// Mitsubishi GX Works2 project: 세척,열풍건조, 동결건조(최신화)   PLC: Q02U

PROGRAM INPUT
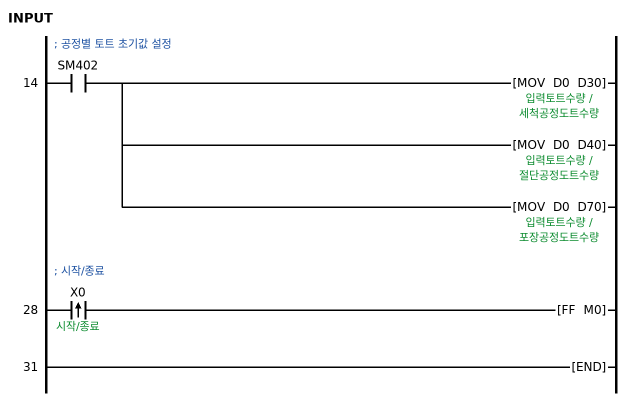
; 공정별 토트 초기값 설정
14    LD      SM402
      MOV     D0 D30  ; 입력토트수량 / 세척공정도트수량
      MOV     D0 D40  ; 절단공정도트수량
      MOV     D0 D70  ; 포장공정도트수량
; 시작/종료
28    LDP     X0  ; 시작/종료
      FF      M0
31    END
END_PROGRAM

PROGRAM 세척공정
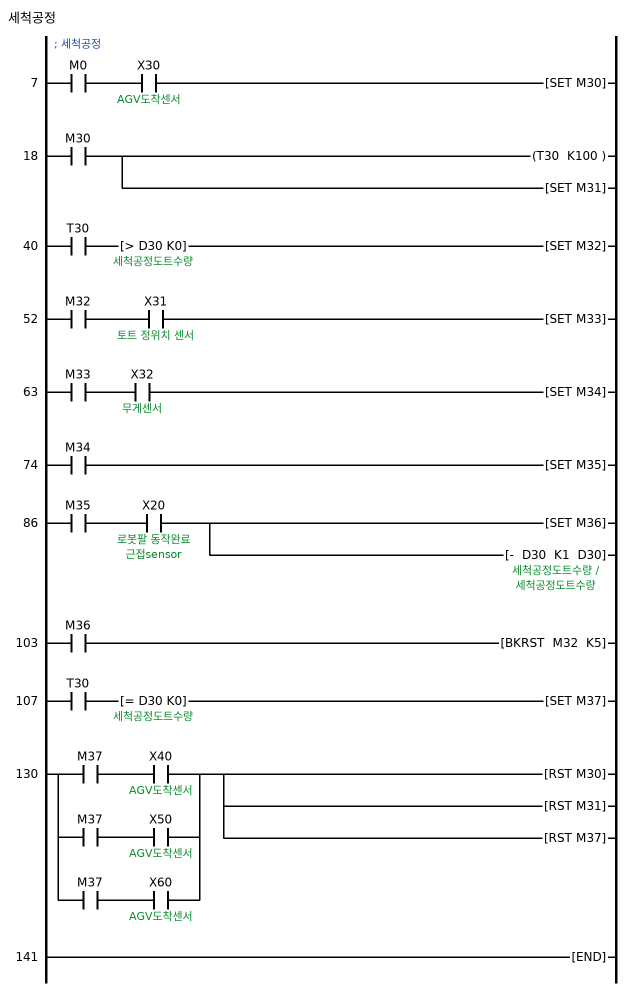
; 세척공정
7     LD      M0
      AND     X30  ; AGV도착센서
      SET     M30
        [note] 펌프모터 ON
18    LD      M30
      OUT     T30 K100
        [note] 펌핑모터 OFF
      SET     M31
        [note] SubCVY ON
40    LD      T30
      AND>    D30 K0  ; 세척공정도트수량
      SET     M32
        [note] 토트 발생
52    LD      M32
      AND     X31  ; 토트 정위치 센서
      SET     M33
        [note] MainCVY ON
63    LD      M33
      AND     X32  ; 무게센서
      SET     M34
        [note] MAinCVY OFF
74    LD      M34
      SET     M35
        [note] 하역 로봇팔 ON
86    LD      M35
      AND     X20  ; 로봇팔 동작완료 근접sensor
      SET     M36
        [note] 하역 로봇팔 OFF
      -       D30 K1 D30
103   LD      M36
      BKRST   M32 K5
107   LD      T30
      AND=    D30 K0  ; 세척공정도트수량
      SET     M37
        [note] AGV 다음 공정 이동, SubCVY OFF
130   LD      M37
      AND     X40  ; AGV도착센서
      LD      M37
      AND     X50  ; AGV도착센서
      ORB
      LD      M37
      AND     X60  ; AGV도착센서
      ORB
      RST     M30
      RST     M31
      RST     M37
141   END
END_PROGRAM

PROGRAM 열풍건조
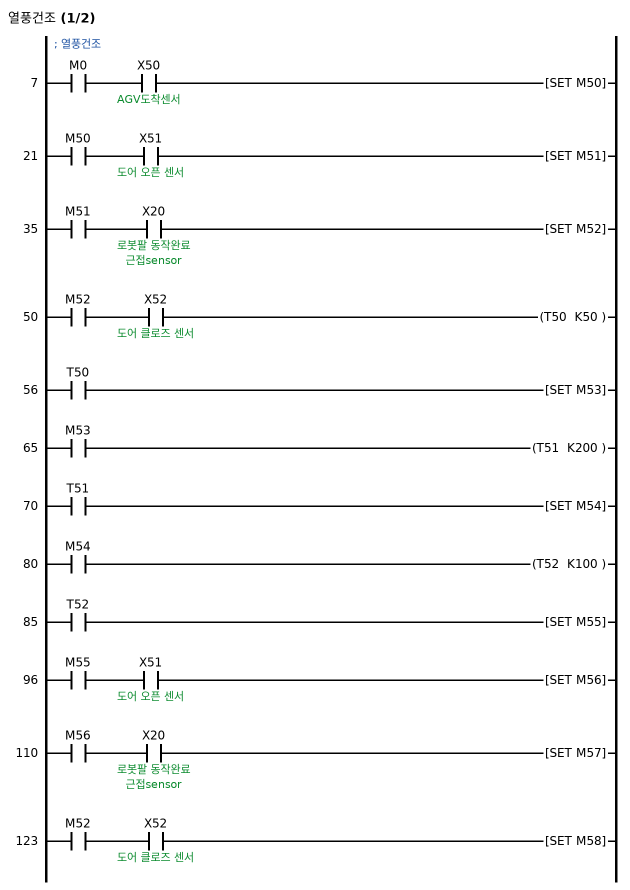
; 열풍건조
7     LD      M0
      AND     X50  ; AGV도착센서
      SET     M50
        [note] 도어 오픈모터(정)
21    LD      M50
      AND     X51  ; 도어 오픈 센서
      SET     M51
        [note] 상역 로봇 팔동작
35    LD      M51
      AND     X20  ; 로봇팔 동작완료 근접sensor
      SET     M52
        [note] 도어 클로즈모터(정)
50    LD      M52
      AND     X52  ; 도어 클로즈 센서
      OUT     T50 K50
56    LD      T50
      SET     M53
        [note] 건조기 ON
65    LD      M53
      OUT     T51 K200
70    LD      T51
      SET     M54
        [note] 건조기 OFF
80    LD      M54
      OUT     T52 K100
85    LD      T52
      SET     M55
        [note] 도어 오픈CYL
96    LD      M55
      AND     X51  ; 도어 오픈 센서
      SET     M56
        [note] 하역 로봇팔 동작
110   LD      M56
      AND     X20  ; 로봇팔 동작완료 근접sensor
      SET     M57
        [note] 도어 클로즈CYL
123   LD      M52
      AND     X52  ; 도어 클로즈 센서
      SET     M58
        [note] AGV 다음 공정 이동
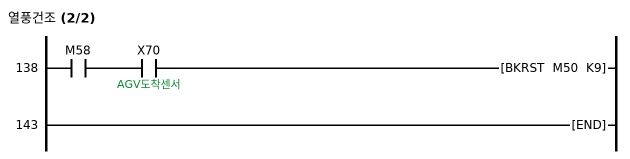
138   LD      M58
      AND     X70  ; AGV도착센서
      BKRST   M50 K9
143   END
END_PROGRAM

PROGRAM OUTPUT
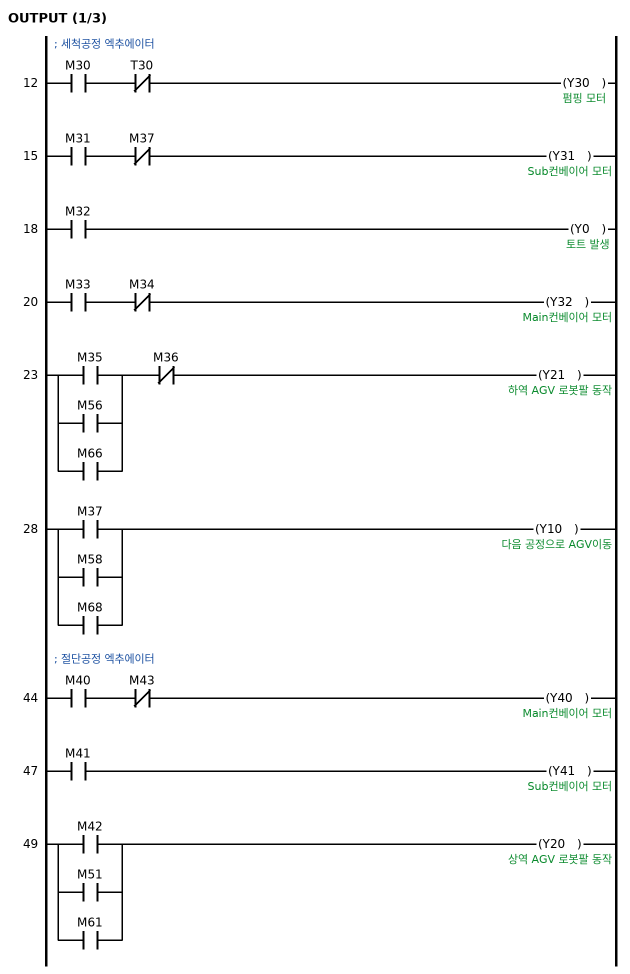
; 세척공정 엑추에이터
12    LD      M30
      ANI     T30
      OUT     Y30  ; 펌핑 모터
15    LD      M31
      ANI     M37
      OUT     Y31  ; Sub컨베이어 모터
18    LD      M32
      OUT     Y0  ; 토트 발생
20    LD      M33
      ANI     M34
      OUT     Y32  ; Main컨베이어 모터
23    LD      M35
      OR      M56
      OR      M66
      ANI     M36
      OUT     Y21  ; 하역 AGV 로봇팔 동작
28    LD      M37
      OR      M58
      OR      M68
      OUT     Y10  ; 다음 공정으로 AGV이동
; 절단공정 엑추에이터
44    LD      M40
      ANI     M43
      OUT     Y40  ; Main컨베이어 모터
47    LD      M41
      OUT     Y41  ; Sub컨베이어 모터
49    LD      M42
      OR      M51
      OR      M61
      OUT     Y20  ; 상역 AGV 로봇팔 동작
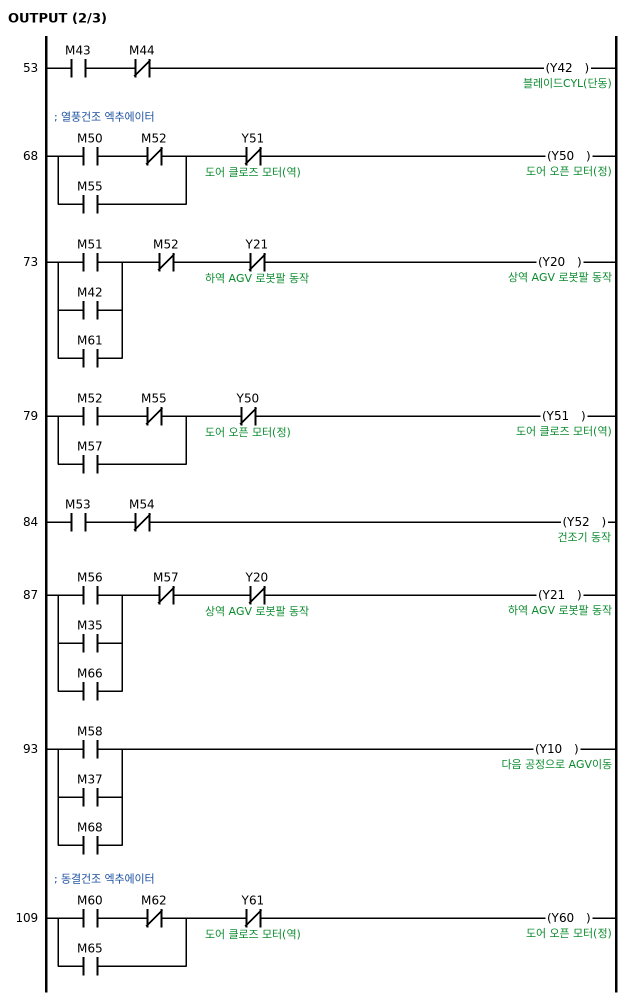
53    LD      M43
      ANI     M44
      OUT     Y42  ; 블레이드CYL(단동)
; 열풍건조 엑추에이터
68    LD      M50
      ANI     M52
      OR      M55
      ANI     Y51  ; 도어 클로즈 모터(역)
      OUT     Y50  ; 도어 오픈 모터(정)
73    LD      M51
      OR      M42
      OR      M61
      ANI     M52
      ANI     Y21  ; 하역 AGV 로봇팔 동작
      OUT     Y20  ; 상역 AGV 로봇팔 동작
79    LD      M52
      ANI     M55
      OR      M57
      ANI     Y50  ; 도어 오픈 모터(정)
      OUT     Y51  ; 도어 클로즈 모터(역)
84    LD      M53
      ANI     M54
      OUT     Y52  ; 건조기 동작
87    LD      M56
      OR      M35
      OR      M66
      ANI     M57
      ANI     Y20  ; 상역 AGV 로봇팔 동작
      OUT     Y21  ; 하역 AGV 로봇팔 동작
93    LD      M58
      OR      M37
      OR      M68
      OUT     Y10  ; 다음 공정으로 AGV이동
; 동결건조 엑추에이터
109   LD      M60
      ANI     M62
      OR      M65
      ANI     Y61  ; 도어 클로즈 모터(역)
      OUT     Y60  ; 도어 오픈 모터(정)
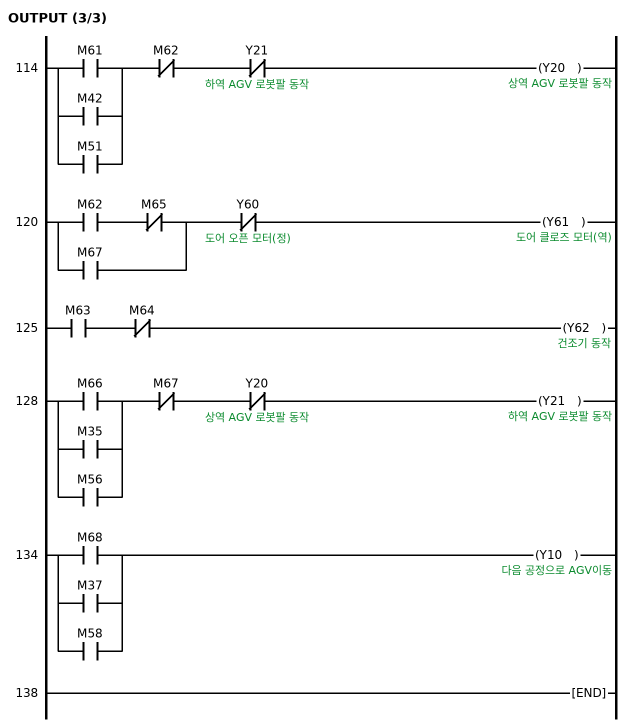
114   LD      M61
      OR      M42
      OR      M51
      ANI     M62
      ANI     Y21  ; 하역 AGV 로봇팔 동작
      OUT     Y20  ; 상역 AGV 로봇팔 동작
120   LD      M62
      ANI     M65
      OR      M67
      ANI     Y60  ; 도어 오픈 모터(정)
      OUT     Y61  ; 도어 클로즈 모터(역)
125   LD      M63
      ANI     M64
      OUT     Y62  ; 건조기 동작
128   LD      M66
      OR      M35
      OR      M56
      ANI     M67
      ANI     Y20  ; 상역 AGV 로봇팔 동작
      OUT     Y21  ; 하역 AGV 로봇팔 동작
134   LD      M68
      OR      M37
      OR      M58
      OUT     Y10  ; 다음 공정으로 AGV이동
138   END
END_PROGRAM

PROGRAM 동결건조
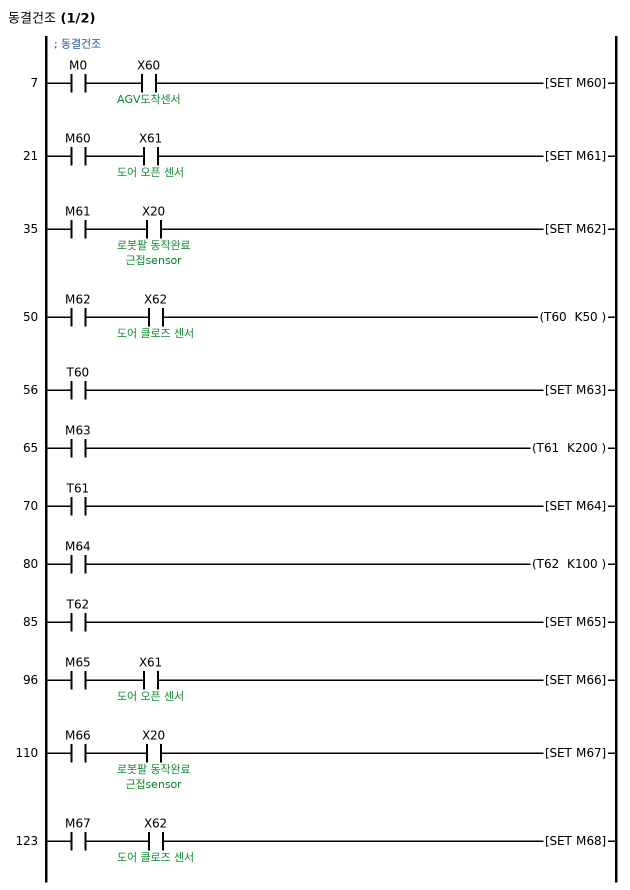
; 동결건조
7     LD      M0
      AND     X60  ; AGV도착센서
      SET     M60
        [note] 도어 오픈모터(정)
21    LD      M60
      AND     X61  ; 도어 오픈 센서
      SET     M61
        [note] 상역 로봇 팔동작
35    LD      M61
      AND     X20  ; 로봇팔 동작완료 근접sensor
      SET     M62
        [note] 도어 클로즈모터(정)
50    LD      M62
      AND     X62  ; 도어 클로즈 센서
      OUT     T60 K50
56    LD      T60
      SET     M63
        [note] 건조기 ON
65    LD      M63
      OUT     T61 K200
70    LD      T61
      SET     M64
        [note] 건조기 OFF
80    LD      M64
      OUT     T62 K100
85    LD      T62
      SET     M65
        [note] 도어 오픈CYL
96    LD      M65
      AND     X61  ; 도어 오픈 센서
      SET     M66
        [note] 하역 로봇팔 동작
110   LD      M66
      AND     X20  ; 로봇팔 동작완료 근접sensor
      SET     M67
        [note] 도어 클로즈CYL
123   LD      M67
      AND     X62  ; 도어 클로즈 센서
      SET     M68
        [note] AGV 다음 공정 이동
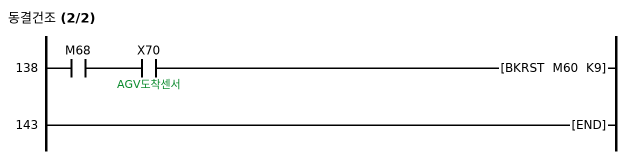
138   LD      M68
      AND     X70  ; AGV도착센서
      BKRST   M60 K9
143   END
END_PROGRAM

PROGRAM 절단공정
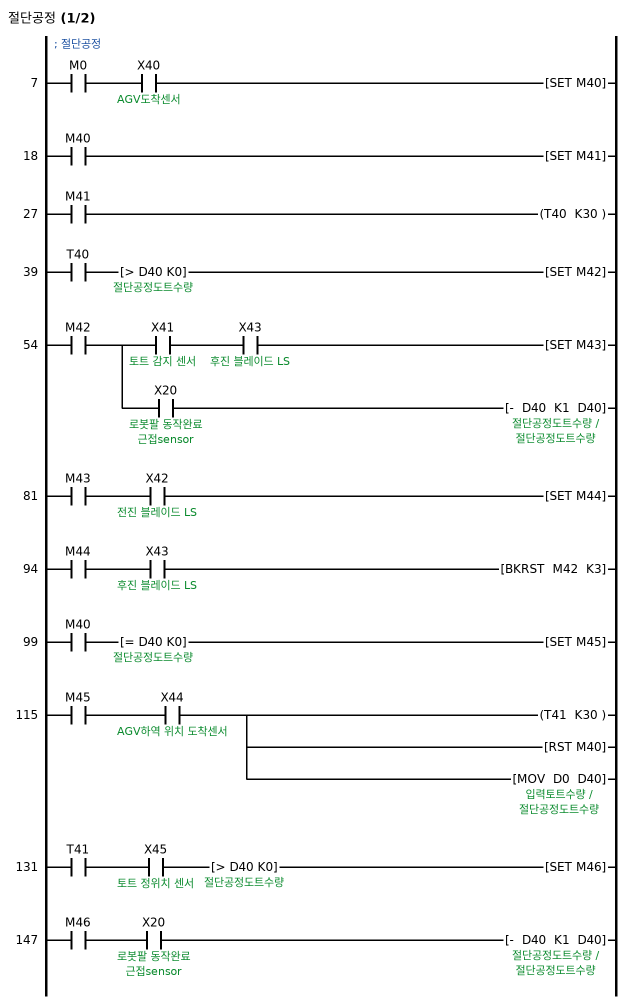
; 절단공정
7     LD      M0
      AND     X40  ; AGV도착센서
      SET     M40
        [note] MainCVY ON
18    LD      M40
      SET     M41
        [note] SubCVY ON
27    LD      M41
      OUT     T40 K30
        [note] 상역 여유
39    LD      T40
      AND>    D40 K0  ; 절단공정도트수량
      SET     M42
        [note] 상역 로봇팔 ON
54    LD      M42
      MPS
      AND     X41  ; 토트 감지 센서
      AND     X43  ; 후진 블레이드 LS
      SET     M43
        [note] MainCVY OFF, 블레이드CYL ON
      MPP
      AND     X20  ; 로봇팔 동작완료 근접sensor
      -       D40 K1 D40
81    LD      M43
      AND     X42  ; 전진 블레이드 LS
      SET     M44
        [note] 블레이드CYL OFF
94    LD      M44
      AND     X43  ; 후진 블레이드 LS
      BKRST   M42 K3
99    LD      M40
      AND=    D40 K0  ; 절단공정도트수량
      SET     M45
        [note] AGV하역 위치 이동
115   LD      M45
      AND     X44  ; AGV하역 위치 도착센서
      OUT     T41 K30
        [note] 하역 여유
      RST     M40
      MOV     D0 D40  ; 입력토트수량
131   LD      T41
      AND     X45  ; 토트 정위치 센서
      AND>    D40 K0  ; 절단공정도트수량
      SET     M46
        [note] 하역 로봇팔 ON
147   LD      M46
      AND     X20  ; 로봇팔 동작완료 근접sensor
      -       D40 K1 D40
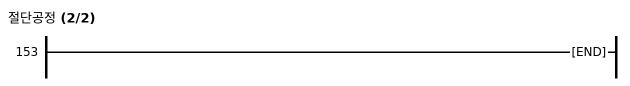
153   END
END_PROGRAM

// device comments not shown above
X12  ; 토틀 감지 센서
D50  ; 열풍건조공정도트수량
D60  ; 동결건조공정도트수량
